# EPICS substitutions: example/exampleApp/Db/example.substitutions
file ADSBIG.template
{
pattern {P, R, PORT, ADDR, TIMEOUT}
	{BL99:Det:, SBIG, S1, 0, 5}
}

file save_restoreStatus.db
{
pattern {P}
        {BL99:CS:SBIG:}
}

file ioc_sns.db
{
pattern {IOCNAME}
        {BL99:CS:SBIG}
}
